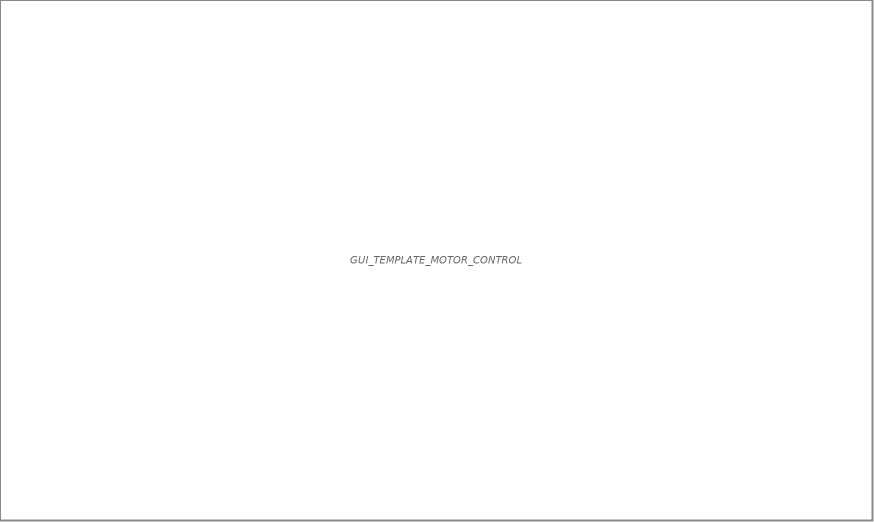
VISUALIZATION GUI_Motor001_Ctrl  // 874x522
    Frame (0,0 872x520)
        shows GUI_TEMPLATE_MOTOR_CONTROL(m_Instance := MAIN.Motor001)
END_VISUALIZATION

(* stored: Version 1.1.0.1, ProductVersion 3.1.4024.3
   Visu GUI_Motor001_Ctrl: Id {ba6b4829-cfe8-4c1b-80a7-d8c3b6d4dc60} *)
